// TwinCAT 3 PLC project TcUnitVerifier
// Title: TcUnit verifier
// Company: www.tcunit.org
// Author: Jakob Sagatowski and other contributors, see CONTRIBUTORS file on www.github.com/tcunit/TcUnit-Verifier
// ProjectVersion: 0.4.1.0
// Description: This project is can be used to verify the different functions of TcUnit. It has various test suites to test different functions in TcUnit. By making sure to comment out everything except the test suite that is interesting it is possible to test only the specific function of TcUnit that is interesting.
// ProgramVersion: 3.1.4022.4
// libraries:
//   Tc2_Standard, * (Beckhoff Automation GmbH)
//   Tc2_System, * (Beckhoff Automation GmbH)
//   Tc3_Module, * (Beckhoff Automation GmbH)
//   TcUnit, * (www.tcunit.org)
// project tree:
//   Mocks/ TestSuiteMock.TcPOU, UnitTestPrinterMock.TcPOU
//   / PlcTask.TcTTO (not stored)
//   Test/ FB_Printer_Test.TcPOU, FB_AnyToUnionValue_Test.TcPOU (not stored), FB_ArrayPrimitiveTypes_Test.TcPOU (not stored), FB_AssertEveryFailedTestTwice.TcPOU (not stored), FB_AssertEveryFailedTestTwice_ArrayVersion.TcPOU (not stored), FB_AssertTrueFalse_Test.TcPOU, FB_CreateFourTestsWithSameName.TcPOU (not stored), FB_CreateDisabledTest.TcPOU (not stored), FB_Runner_Test.TcPOU, FB_PrimitiveTypes_Test.TcPOU (not stored), FB_AnyPrimitiveTypes_Test.TcPOU (not stored), FB_SimpleStringBuilder_Test.TcPOU, FB_AnyToString_Test.TcPOU, FB_TestSuite_Test.TcPOU, PRG_TEST.TcPOU

// ---- Mocks/TestSuiteMock.TcPOU
FUNCTION_BLOCK TestSuiteMock EXTENDS UnitTestSuite IMPLEMENTS ITestSuite
VAR_INPUT
END_VAR
VAR_OUTPUT
END_VAR
VAR
    runTestsCounter: UINT := 0;
END_VAR

METHOD runAllTests
runTestsCounter := runTestsCounter + 1;
END_METHOD

PROPERTY runAllTestsExecuted : BOOL
GET
runAllTestsExecuted := runTestsCounter > 0;
END_GET
END_PROPERTY

END_FUNCTION_BLOCK

// ---- Mocks/UnitTestPrinterMock.TcPOU
FUNCTION_BLOCK UnitTestPrinterMock EXTENDS UnitTestPrinter
VAR_INPUT
END_VAR
VAR_OUTPUT
END_VAR
VAR
END_VAR

METHOD getFailMessage : MaxString
VAR_INPUT
END_VAR
getFailMessage := messageBuilder.toString();
END_METHOD

END_FUNCTION_BLOCK

// ---- Test/FB_Printer_Test.TcPOU
{attribute 'call_after_init'}
FUNCTION_BLOCK FB_Printer_Test EXTENDS TcUnit.FB_TestSuite IMPLEMENTS TcUnit.I_RunnableTestSuite
VAR
    Assert : TcUnit.FB_Assert;
    
    getFailureMessageString_Printer: UnitTestPrinter;
    getFailureMessageINT_Printer: UnitTestPrinter;
END_VAR

METHOD FB_init : BOOL
VAR_INPUT
	bInitRetains : BOOL; // if TRUE, the retain variables are initialized (warm start / cold start)
	bInCopyCode : BOOL;  // if TRUE, the instance afterwards gets moved into the copy code (online change)
END_VAR
SUPER^.RegisterTestSuite(THIS^);
END_METHOD

METHOD RunTests : TCUNIT.E_TestSuiteRunState
Test_GetFailureMessageString();
Test_GetFailureMessageINT();

RunTests := TCUNIT.E_TestSuiteRunState.FINISHED;
END_METHOD

METHOD Test_GetFailureMessageINT
VAR
    expected: MaxString;
    actual: MaxString;
    
    expectedTestValue: INT;
    actualTestValue: INT;
    message: MaxString;
    path: MaxString;
END_VAR
TEST('Test_GetFailureMessageINT');

expected := 'FAILED TEST $'FB_TestSuite_Test$', EXP: 1234, ACT: 1235, MSG: INTs do not match';

expectedTestValue := 1234;
actualTestValue := 1235;
message := 'INTs do not match';
path := 'FB_TestSuite_Test';
actual := getFailureMessageINT_Printer.getFailureMessage(expectedTestValue, actualTestValue, message, path);

Assert.AssertEquals_STRING(expected, actual, 'Get Failure Message INT does not match');
END_METHOD

METHOD Test_GetFailureMessageString
VAR
    expected: MaxString;
    actual: MaxString;
    
    expectedTestValue: MaxString;
    actualTestValue: MaxString;
    message: MaxString;
    path: MaxString;
END_VAR
TEST('Test_GetFailureMessageString');

expected := 'FAILED TEST $'FB_TestSuite_Test$', EXP: hello, ACT: world, MSG: Strings do not match';

expectedTestValue := 'hello';
actualTestValue := 'world';
message := 'Strings do not match';
path := 'FB_TestSuite_Test';
actual := getFailureMessageString_Printer.getFailureMessage(expectedTestValue, actualTestValue, message, path);

Assert.AssertEquals_STRING(expected, actual, 'Get Failure Message String does not match');
END_METHOD

END_FUNCTION_BLOCK

// ---- Test/FB_TestSuite_Test.TcPOU
{attribute 'call_after_init'}
FUNCTION_BLOCK FB_TestSuite_Test EXTENDS TcUnit.FB_TestSuite IMPLEMENTS TcUnit.I_RunnableTestSuite
VAR
    Assert : TcUnit.FB_Assert;

    numberOfTestsZero_TestSuite: UnitTestSuite(0);

    testSuiteRegistersItself_Runner: UnitTestRunner;
    testSuiteRegistersItself_TestSuite: UnitTestSuite(testSuiteRegistersItself_Runner);
    
    runAllTestsWithOneTestSuite_Runner: UnitTestRunner;
    runAllTestsWithOneTestSuite_TestSuite: TestSuiteMock(runAllTestsWithOneTestSuite_Runner);
    
    runAllTestsWithFourTestSuites_Runner: UnitTestRunner;
    runAllTestsWithFourTestSuites_TestSuite1: TestSuiteMock(runAllTestsWithFourTestSuites_Runner);
    runAllTestsWithFourTestSuites_TestSuite2: TestSuiteMock(runAllTestsWithFourTestSuites_Runner);
    runAllTestsWithFourTestSuites_TestSuite3: TestSuiteMock(runAllTestsWithFourTestSuites_Runner);
    runAllTestsWithFourTestSuites_TestSuite4: TestSuiteMock(runAllTestsWithFourTestSuites_Runner);
END_VAR

METHOD FB_init : BOOL
VAR_INPUT
	bInitRetains : BOOL; // if TRUE, the retain variables are initialized (warm start / cold start)
	bInCopyCode : BOOL;  // if TRUE, the instance afterwards gets moved into the copy code (online change)
END_VAR
SUPER^.RegisterTestSuite(THIS^);
END_METHOD

METHOD RunTests : TCUNIT.E_TestSuiteRunState
Test_NumberOfTestsZero();
Test_TestSuiteRegistersItself();
Test_RunAllTestsWithOneTestSuite();
Test_RunAllTestsWithFourTestSuites();

RunTests := TCUNIT.E_TestSuiteRunState.FINISHED;
END_METHOD

METHOD Test_NumberOfTestsZero
VAR
    expected: UINT;
    actual: UINT;
END_VAR
TEST('Test_NumberOfTestsZero');

expected := 0;
actual := numberOfTestsZero_TestSuite.numberOfTests;

Assert.AssertEquals_UINT(expected, actual, 'Number of Tests is non zero');
END_METHOD

METHOD Test_RunAllTestsWithFourTestSuites
VAR
    expected: BOOL;
    actual: BOOL;
END_VAR
TEST('Test_RunAllTestsWithFourTestSuites');

runAllTestsWithFourTestSuites_Runner.runAllTests();

expected := TRUE;
actual := runAllTestsWithFourTestSuites_TestSuite1.runAllTestsExecuted;
actual := actual AND runAllTestsWithFourTestSuites_TestSuite2.runAllTestsExecuted;
actual := actual AND runAllTestsWithFourTestSuites_TestSuite3.runAllTestsExecuted;
actual := actual AND runAllTestsWithFourTestSuites_TestSuite4.runAllTestsExecuted;

Assert.AssertEquals_BOOL(expected, actual, 'Test Suite not executed even though the runner ran');
END_METHOD

METHOD Test_RunAllTestsWithOneTestSuite
VAR
    expected: BOOL;
    actual: BOOL;
END_VAR
TEST('Test_RunAllTestsWithOneTestSuite');

expected := FALSE;
actual := runAllTestsWithOneTestSuite_TestSuite.runAllTestsExecuted;

Assert.AssertEquals_BOOL(expected, actual, 'Test Suite executed even though the runner did not run');

runAllTestsWithOneTestSuite_Runner.runAllTests();

expected := TRUE;
actual := runAllTestsWithOneTestSuite_TestSuite.runAllTestsExecuted;

Assert.AssertEquals_BOOL(expected, actual, 'Test Suite not executed even though the runner ran');
END_METHOD

METHOD Test_TestSuiteRegistersItself
VAR
    expected: UINT;
    actual: UINT;
END_VAR
TEST('Test_TestSuiteRegistersItself');

expected := 1;
actual := testSuiteRegistersItself_Runner.numberOfTestSuites;

Assert.AssertEquals_UINT(expected, actual, 'Test Suite did not register itself');
END_METHOD

END_FUNCTION_BLOCK

// ---- Test/FB_AssertTrueFalse_Test.TcPOU
(* 
    This testsuite verifies that the Assert_True and Assert_False methods do what they are supposed to. It does so
    by making sure that every assert-method (assert_true & assert_false) does both one failing and one successful
    assert.
*)
{attribute 'call_after_init'}
FUNCTION_BLOCK FB_AssertTrueFalse_Test EXTENDS TcUnit.FB_TestSuite IMPLEMENTS TcUnit.I_RunnableTestSuite
VAR
    Assert : TcUnit.FB_Assert;
END_VAR

METHOD PRIVATE AssertThatINTsAreEqual
VAR
    a : INT := -33;
    b : INT := -44;
END_VAR
TEST('AssertThatINTsAreEqual');

Assert.AssertFalse(Condition := (a <> b),
                   Message := 'INTs are equal');
END_METHOD

METHOD PRIVATE AssertThatINTsAreNotEqual
VAR
    a : INT := -33;
    b : INT := -44;
END_VAR
TEST('AssertThatINTsAreNotEqual');

Assert.AssertFalse(Condition := (a = b),
                   Message := 'INTs are equal');
END_METHOD

METHOD PRIVATE AssertThatWORDsAreEqual
VAR
    a : WORD := 16#ABCD;
    b : WORD := 16#0123;
END_VAR
TEST('AssertThatWORDsAreEqual');

Assert.AssertTrue(Condition := (a = b),
                  Message := 'WORDs are not equal');
END_METHOD

METHOD PRIVATE AssertThatWORDsAreNotEqual
VAR
    a : WORD := 16#ABCD;
    b : WORD := 16#0123;
END_VAR
TEST('AssertThatWORDsAreNotEqual');

Assert.AssertTrue(Condition := (a <> b),
                  Message := 'WORDs are equal');
END_METHOD

METHOD FB_init : BOOL
VAR_INPUT
	bInitRetains : BOOL; // if TRUE, the retain variables are initialized (warm start / cold start)
	bInCopyCode : BOOL;  // if TRUE, the instance afterwards gets moved into the copy code (online change)
END_VAR
SUPER^.RegisterTestSuite(THIS^);
END_METHOD

METHOD RunTests : TCUNIT.E_TestSuiteRunState
AssertThatINTsAreEqual();
AssertThatINTsAreNotEqual();
AssertThatWORDsAreEqual();
AssertThatWORDsAreNotEqual();

RunTests := TCUNIT.E_TestSuiteRunState.FINISHED;
END_METHOD

END_FUNCTION_BLOCK

// ---- Test/FB_Runner_Test.TcPOU
{attribute 'call_after_init'}
FUNCTION_BLOCK FB_Runner_Test EXTENDS TcUnit.FB_TestSuite IMPLEMENTS TcUnit.I_RunnableTestSuite
VAR
    Assert : TcUnit.FB_Assert;
    
    numberOfTestSuitesZero_Runner: UnitTestRunner;
    
    numberOfTestSuitesOne_Runner: UnitTestRunner;
    numberOfTestSuitesOne_TestSuite: UnitTestSuite(0);
    
    numberOfTestSuitesThree_Runner: UnitTestRunner;
    numberOfTestSuitesThree_TestSuite1: UnitTestSuite(0);
    numberOfTestSuitesThree_TestSuite2: UnitTestSuite(0);
    numberOfTestSuitesThree_TestSuite3: UnitTestSuite(0);
    
    sameTestSuiteCountsAsOne_Runner: UnitTestRunner;
    sameTestSuiteCountsAsOne_TestSuite: UnitTestSuite(0);
END_VAR

METHOD FB_init : BOOL
VAR_INPUT
	bInitRetains : BOOL; // if TRUE, the retain variables are initialized (warm start / cold start)
	bInCopyCode : BOOL;  // if TRUE, the instance afterwards gets moved into the copy code (online change)
END_VAR
SUPER^.RegisterTestSuite(THIS^);
END_METHOD

METHOD RunTests : TCUNIT.E_TestSuiteRunState
Test_NumberOfTestSuitesZero();
Test_NumberOfTestSuitesOne();
Test_NumberOfTestSuitesThree();
Test_SameTestSuiteCountsAsOne();

RunTests := TCUNIT.E_TestSuiteRunState.FINISHED;
END_METHOD

METHOD Test_NumberOfTestSuitesOne
VAR
    expected: UINT;
    actual: UINT;
END_VAR
TEST('Test_NumberOfTestSuitesOne');

expected := 1;
numberOfTestSuitesOne_Runner.registerTestSuite(numberOfTestSuitesOne_TestSuite);
actual := numberOfTestSuitesOne_Runner.numberOfTestSuites;

Assert.AssertEquals_UINT(expected, actual, 'Number of Runner Test Suites unequal one');
END_METHOD

METHOD Test_NumberOfTestSuitesThree
VAR
    expected: UINT;
    actual: UINT;
END_VAR
TEST('Test_NumberOfTestSuitesThree');

expected := 3;
numberOfTestSuitesThree_Runner.registerTestSuite(numberOfTestSuitesThree_TestSuite1);
numberOfTestSuitesThree_Runner.registerTestSuite(numberOfTestSuitesThree_TestSuite2);
numberOfTestSuitesThree_Runner.registerTestSuite(numberOfTestSuitesThree_TestSuite3);
actual := numberOfTestSuitesThree_Runner.numberOfTestSuites;

Assert.AssertEquals_UINT(expected, actual, 'Number of Runner Test Suites unequal three');
END_METHOD

METHOD Test_NumberOfTestSuitesZero
VAR
    expected: UINT;
    actual: UINT;
END_VAR
TEST('Test_NumberOfTestSuitesZero');

expected := 0;
actual := numberOfTestSuitesZero_Runner.numberOfTestSuites;

Assert.AssertEquals_UINT(expected, actual, 'Number of Runner Test Suites unequal zero');
END_METHOD

METHOD Test_SameTestSuiteCountsAsOne
VAR
    expected: UINT;
    actual: UINT;
END_VAR
TEST('Test_SameTestSuiteCountsAsOne');

expected := 1;
sameTestSuiteCountsAsOne_Runner.registerTestSuite(sameTestSuiteCountsAsOne_TestSuite);
sameTestSuiteCountsAsOne_Runner.registerTestSuite(sameTestSuiteCountsAsOne_TestSuite);
actual := sameTestSuiteCountsAsOne_Runner.numberOfTestSuites;

Assert.AssertEquals_UINT(expected, actual, 'Same Test Suite should not be counted more than once');
END_METHOD

END_FUNCTION_BLOCK

// ---- Test/FB_SimpleStringBuilder_Test.TcPOU
{attribute 'call_after_init'}
FUNCTION_BLOCK FB_SimpleStringBuilder_Test EXTENDS TcUnit.FB_TestSuite IMPLEMENTS TcUnit.I_RunnableTestSuite
VAR
    Assert : TcUnit.FB_Assert;
    
    initializedStringBuilderEmpty_StringBuilder: SimpleStringBuilder;
    
    appendOneString_StringBuilder: SimpleStringBuilder;
    
    appendThreeStrings_StringBuilder: SimpleStringBuilder;
    
    appendINT_StringBuilder: SimpleStringBuilder;
END_VAR

METHOD FB_init : BOOL
VAR_INPUT
	bInitRetains : BOOL; // if TRUE, the retain variables are initialized (warm start / cold start)
	bInCopyCode : BOOL;  // if TRUE, the instance afterwards gets moved into the copy code (online change)
END_VAR
SUPER^.RegisterTestSuite(THIS^);
END_METHOD

METHOD RunTests : TCUNIT.E_TestSuiteRunState
Test_InitializedStringBuilderEmpty();
Test_AppendOneString();
Test_AppendThreeStrings();
Test_AppendINT();

RunTests := TCUNIT.E_TestSuiteRunState.FINISHED;
END_METHOD

METHOD Test_AppendINT
VAR
    expected: STRING(10);
    actual: STRING(10);
    
    testINT: INT;
END_VAR
TEST('Test_AppendINT');

expected := '13';

testINT := 13;
appendINT_StringBuilder.append(testINT);
actual := appendINT_StringBuilder.toString();

Assert.AssertEquals_STRING(expected, actual, 'Appended INT does not match');
END_METHOD

METHOD Test_AppendOneString
VAR
    expected: STRING(10);
    actual: STRING(10);
    
    testString: STRING(10);
END_VAR
TEST('Test_AppendOneString');

expected := 'twincat$R';

testString := 'twincat$R';
appendOneString_StringBuilder.append(testString);
actual := appendOneString_StringBuilder.toString();

Assert.AssertEquals_STRING(expected, actual, 'String did not append');
END_METHOD

METHOD Test_AppendThreeStrings
VAR
    expected: STRING(30);
    actual: STRING(30);
    
    testString1: STRING(10);
    testString2: STRING(10);
    testString3: STRING(10);
END_VAR
TEST('Test_AppendThreeStrings');

expected := 'hello$Tworld$Tfoo$R';

testString1 := 'hello$T';
appendThreeStrings_StringBuilder.append(testString1);
testString2 := 'world$T';
appendThreeStrings_StringBuilder.append(testString2);
testString3 := 'foo$R';
appendThreeStrings_StringBuilder.append(testString3);
actual := appendThreeStrings_StringBuilder.toString();

Assert.AssertEquals_STRING(expected, actual, 'Appended Strings do not match');
END_METHOD

METHOD Test_InitializedStringBuilderEmpty
VAR
    expected: STRING(10);
    actual: STRING(10);
END_VAR
TEST('Test_InitializedStringBuilderEmpty');

expected := '';
actual := initializedStringBuilderEmpty_StringBuilder.toString();

Assert.AssertEquals_STRING(expected, actual, 'Initialized String Builder not empty');
END_METHOD

END_FUNCTION_BLOCK

// ---- Test/FB_AnyToString_Test.TcPOU
{attribute 'call_after_init'}
FUNCTION_BLOCK FB_AnyToString_Test EXTENDS TcUnit.FB_TestSuite IMPLEMENTS TcUnit.I_RunnableTestSuite
VAR
    Assert : TcUnit.FB_Assert;
END_VAR

METHOD FB_init : BOOL
VAR_INPUT
	bInitRetains : BOOL; // if TRUE, the retain variables are initialized (warm start / cold start)
	bInCopyCode : BOOL;  // if TRUE, the instance afterwards gets moved into the copy code (online change)
END_VAR
SUPER^.RegisterTestSuite(THIS^);
END_METHOD

METHOD RunTests : TCUNIT.E_TestSuiteRunState
Test_String();
Test_INT();
Test_REAL();

RunTests := TCUNIT.E_TestSuiteRunState.FINISHED;
END_METHOD

METHOD Test_INT
VAR
    expected: STRING(10);
    actual: STRING(10);
    
    testINT: INT;
END_VAR
TEST('Test_INT');

expected := '1001';

testINT := 1001;
actual := anyToString(testINT);

Assert.AssertEquals_STRING(expected, actual, 'Any INT does not match');
END_METHOD

METHOD Test_REAL
VAR
    expected: STRING(10);
    actual: STRING(10);
    
    testREAL: REAL;
END_VAR
TEST('Test_REAL');

expected := '13.789';

testREAL := 13.789;
actual := anyToString(testREAL);

Assert.AssertEquals_STRING(expected, actual, 'Any REAL does not match');
END_METHOD

METHOD Test_String
VAR
    expected: STRING(10);
    actual: STRING(10);
END_VAR
TEST('Test_String');

expected := 'hello';

actual := anyToString(expected);

Assert.AssertEquals_STRING(expected, actual, 'Any String does not match');
END_METHOD

END_FUNCTION_BLOCK

// ---- Test/PRG_TEST.TcPOU
PROGRAM PRG_TEST
VAR
    (*PrimitiveTypesTest : FB_PrimitiveTypes_Test;
    AssertTrueFalse_Test : FB_AssertTrueFalse_Test;
    AssertEveryFailedTestTwice : FB_AssertEveryFailedTestTwice;
    CreateFourTestsWithSameName : FB_CreateFourTestsWithSameName;
    ArrayPrimitiveTypes_Test : FB_ArrayPrimitiveTypes_Test;
    CreateDisabledTest : FB_CreateDisabledTest;
    AnyPrimitiveTypes_Test : FB_AnyPrimitiveTypes_Test;
    AssertEveryFailedTestTwice_ArrayVersion : FB_AssertEveryFailedTestTwice_ArrayVersion;
    AnyToUnionValue_Test : FB_AnyToUnionValue_Test;*)
    AnyToString_Test: FB_AnyToString_Test;
    SimpleStringBuilder_Test: FB_SimpleStringBuilder_Test;
    Printer_Test: FB_Printer_Test;
    Runner_Test: FB_Runner_Test;
    TestSuite_Test: FB_TestSuite_Test;
END_VAR

TcUnit.RUN();

END_PROGRAM
